// Mitsubishi GX Works2 project: PLC_Group5   PLC: FX3G

// global labels: Global1
VAR_GLOBAL
  Start_DAY AT X007 : BOOL;
  Lamp_Start_Internal AT M7 : BOOL;
END_VAR
VAR_GLOBAL CONSTANT
  Min_Protein : REAL := 320.0;
  Min_Oat : REAL := 400;
  Min_honey : REAL := 160.0;
END_VAR
VAR_GLOBAL
  End_Triger AT X005 : BOOL;
  End_Day AT M3 : BOOL;
  START_Day_Lamp AT X007 : BOOL;
  End_Day_Lamp AT X007 : BOOL;
  Lamp_Start_initaal AT M1 : BOOL;
  Day_Work_Lamp AT Y000 : BOOL;
  Mix_Products AT X003 : BOOL;
  Anlog_Inpute AT D8280 : INT;
END_VAR
VAR_GLOBAL CONSTANT
  Min_Analog : REAL := 5.0;
END_VAR
VAR_GLOBAL
  Save AT X007 : BOOL;
END_VAR
VAR_GLOBAL CONSTANT
  Max_Analog : REAL := 5;
END_VAR
VAR_GLOBAL
  Save_Anlog_Classic AT D8282 : INT;
  Save_Anlog_Protein AT D8282 : INT;
  Save_Lamp_Input AT M1 : BOOL;
END_VAR
VAR_GLOBAL CONSTANT
  Constant_400 : REAL := 400;
END_VAR
VAR_GLOBAL
  Normalized_Inpute AT M20 : BOOL;
  Input_Hone AT D1150 : REAL;
  M_hone AT D1152 : REAL;
  Input_Oat AT D1154 : REAL;
  M_Oat AT D1156 : REAL;
  Input_Protein AT D1158 : REAL;
  M_Protein AT D1160 : REAL;
  M_PM_Proteinrotein AT D1160 : REAL;
  Input_Ans AT D1302 : REAL;
  USER_PICK AT D1300 : REAL;
  Classic AT M22 : BOOL;
  Protein AT M23 : BOOL;
END_VAR
VAR_GLOBAL CONSTANT
  LessHone_120 : REAL := 120.0;
  LessOat_400 : REAL := 400.0;
  Less_Protien_160 : REAL := 160.0;
  LessOat_240 : REAL := 240.0;
  LessHone_160 : REAL := 160.0;
  LessProtien_320 : REAL := 320.0;
  LessHone_15 : REAL := 15.0;
  LessOat_50 : REAL := 50.0;
  Less_Protien_20 : REAL := 20.0;
  LessHone_20 : REAL := 20.0;
  LessOat_30 : REAL := 30.0;
  LessProtien_40 : REAL := 40.0;
END_VAR
VAR_GLOBAL
  Timer_MIX AT TC10 : BOOL;
END_VAR
VAR_GLOBAL CONSTANT
  Time_value : WORD := 50;
END_VAR
VAR_GLOBAL
  Lamp_MIX AT Y003 : BOOL;
  Start_baking AT X002 : BOOL;
  Blink_Lamp AT M30 : BOOL;
  Timer_Bake_Clasicc AT TC2 : BOOL;
END_VAR
VAR_GLOBAL CONSTANT
  Bakt_TimeClassic : WORD := 4;
END_VAR
VAR_GLOBAL
  Ts1 AT TC2 : BOOL;
  Baking_Lamp1 AT Y001 : BOOL;
  Timer_Bake_Protein AT TC3 : BOOL;
  Ts2 AT TC3 : BOOL;
  Baking_Lamp2 AT Y002 : BOOL;
  Start_packing AT X006 : BOOL;
  Add_Snack AT X000 : BOOL;
  Packing_Lamp AT Y004 : BOOL;
  Snack_Num AT CC1 : BOOL;
END_VAR
VAR_GLOBAL CONSTANT
  BOX : WORD := 1;
END_VAR
VAR_GLOBAL
  CS AT CS1 : BOOL;
  StoringSnacks AT X002 : BOOL;
END_VAR
VAR_GLOBAL CONSTANT
  Add_1 : REAL := 1.0;
  Div_analog2 : REAL := 40;
END_VAR
VAR_GLOBAL
  Num_of_Snacks_Packs AT D1202 : REAL;
  Analog_Output AT D8282 : INT;
  Protein_chose AT M23 : BOOL;
  Protein_chosen AT CC23 : BOOL;
  Classic_chosen AT CC22 : BOOL;
  Classic_1 AT M82 : BOOL;
  Protein_1 AT M89 : BOOL;
  Blinking_Lamp AT M33 : BOOL;
  Timer_Bake_One AT TC2 : BOOL;
  Timer_Bake_Two AT TC3 : BOOL;
END_VAR
VAR_GLOBAL CONSTANT
  TimeForCS : WORD := 30;
  TimeForPS : WORD := 60;
END_VAR
VAR_GLOBAL
  Flash_Count AT TC5 : BOOL;
  Bake_Time AT D5000 : WORD;
  CountFirst_Snack_Num AT CC1 : BOOL;
END_VAR
VAR_GLOBAL CONSTANT
  FirstBar : WORD := 1;
END_VAR
VAR_GLOBAL
  One_Bar_Count AT CS1 : BOOL;
  Seven_Bar_Count AT CS2 : BOOL;
  Count_7_bars AT CC2 : BOOL;
END_VAR
VAR_GLOBAL CONSTANT
  SevenBar : WORD := 8;
END_VAR
VAR_GLOBAL
  Snack_Storage AT D1202 : REAL;
  Stock_Check AT M50 : BOOL;
  StockStock_Check_Check AT M50 : BOOL;
END_VAR
VAR_GLOBAL CONSTANT
  ResAnalogOutput : INT;
  ZeroHone : REAL;
  ZeroOat : REAL;
  ZeroProtein : REAL;
END_VAR

// task Task_01 (event TRUE, interval 0, priority 31): POU_01

PROGRAM POU_01
(* structured ladder/FBD written out as ST: instructions are called as NAME(EN, inputs, outputs); _pN, _eN, _tN stand for wires *)
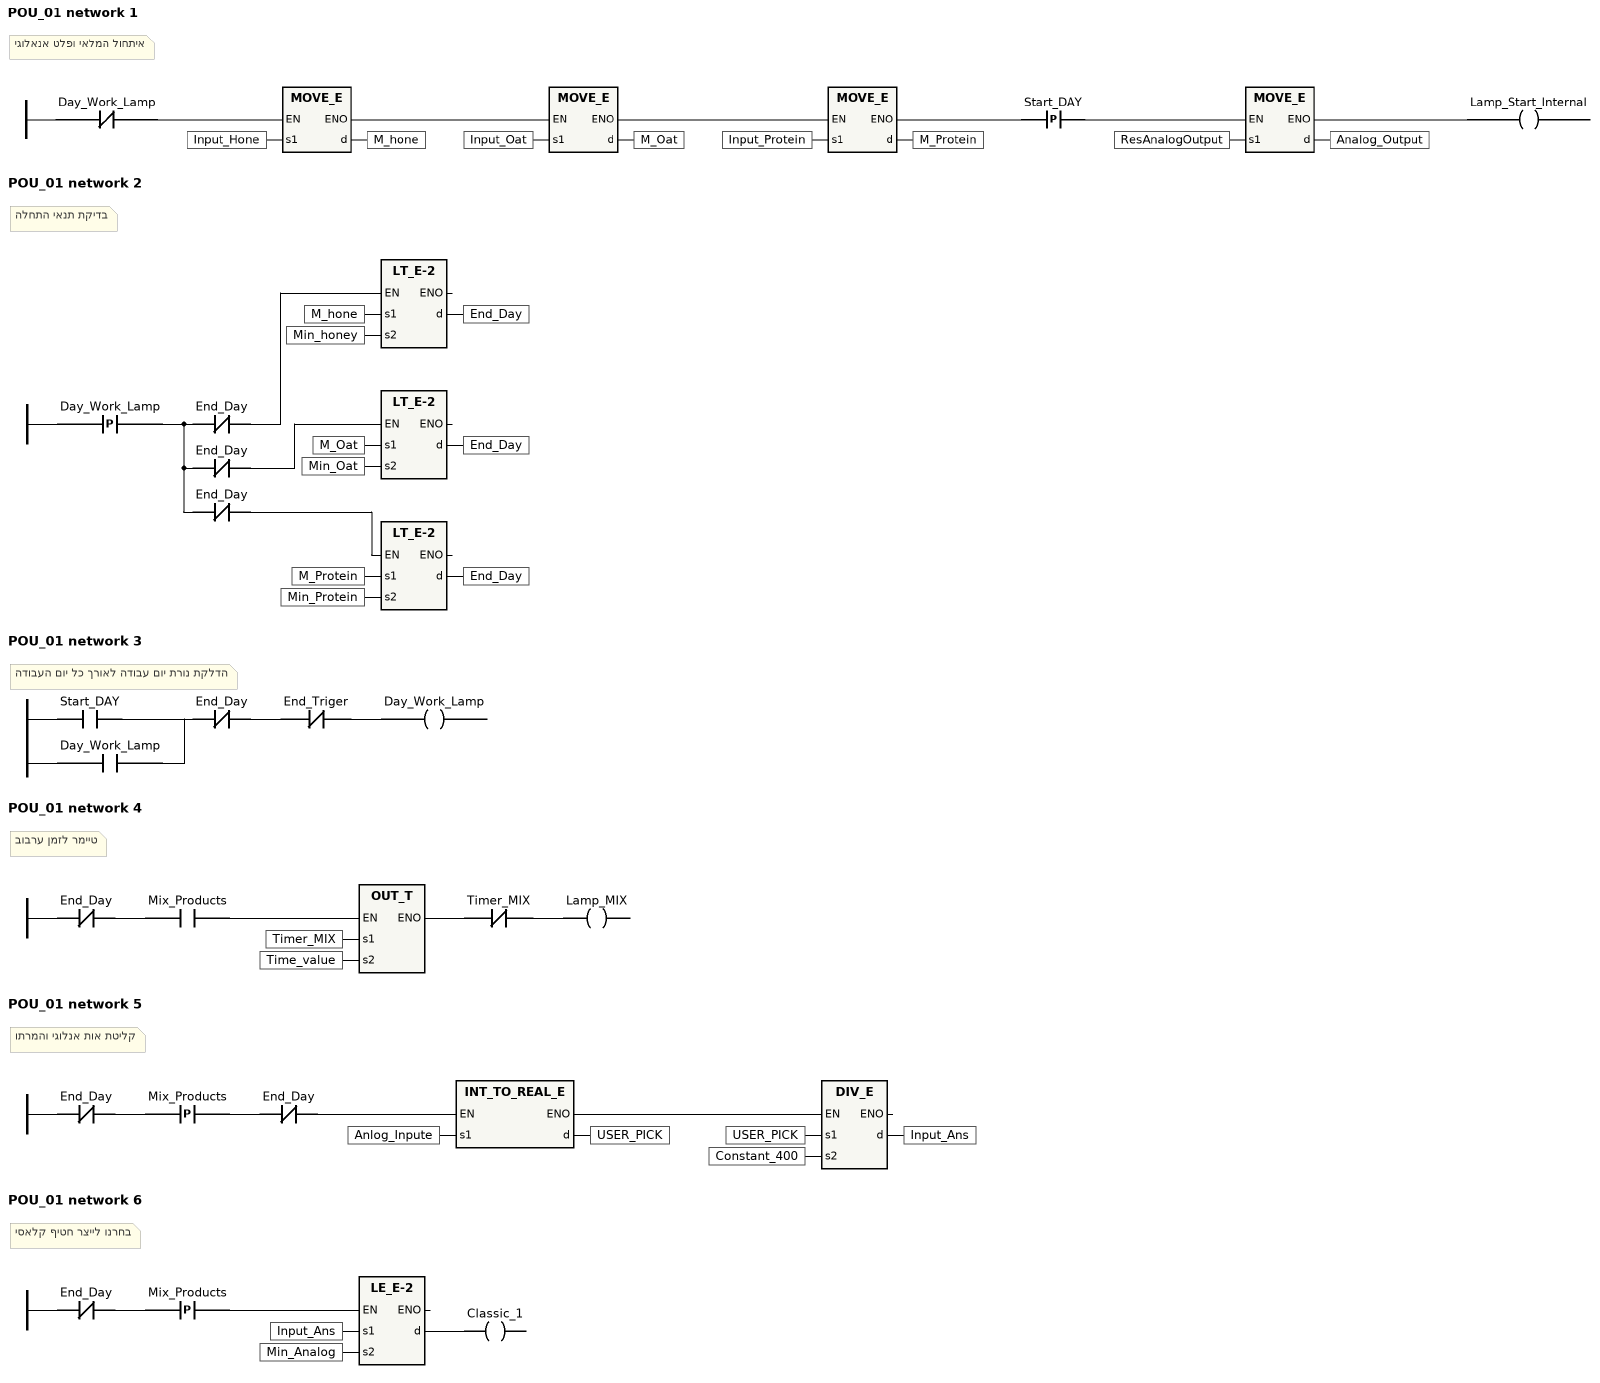
(* network 1 *)
(* איתחול המלאי ופלט אנאלוגי *)
_e1 := MOVE_E(NOT Day_Work_Lamp, Input_Hone, M_hone);
_e2 := MOVE_E(_e1, Input_Oat, M_Oat);
_e3 := MOVE_E(_e2, Input_Protein, M_Protein);
_e4 := MOVE_E(_e3 AND LDP(TRUE, Start_DAY), ResAnalogOutput, Analog_Output);
Lamp_Start_Internal := _e4;
(* network 2 *)
(* בדיקת תנאי התחלה *)
_p1 := LDP(TRUE, Day_Work_Lamp);
LT_E(_p1 AND NOT End_Day, M_hone, Min_honey, End_Day);
LT_E(_p1 AND NOT End_Day, M_Oat, Min_Oat, End_Day);
LT_E(_p1 AND NOT End_Day, M_Protein, Min_Protein, End_Day);
(* network 3 *)
(* הדלקת נורת יום עבודה לאורך כל יום העבודה *)
Day_Work_Lamp := ((Start_DAY OR Day_Work_Lamp) AND NOT End_Day) AND NOT End_Triger;
(* network 4 *)
(* טיימר לזמן ערבוב *)
_e1 := OUT_T(NOT End_Day AND Mix_Products, Timer_MIX, Time_value);
Lamp_MIX := _e1 AND NOT Timer_MIX;
(* network 5 *)
(* קליטת אות אנלוגי והמרתו *)
_e1 := INT_TO_REAL_E(NOT End_Day AND LDP(TRUE, Mix_Products) AND NOT End_Day, Anlog_Inpute, USER_PICK);
DIV_E(_e1, USER_PICK, Constant_400, Input_Ans);
(* network 6 *)
(* בחרנו לייצר חטיף קלאסי *)
LE_E(NOT End_Day AND LDP(TRUE, Mix_Products), Input_Ans, Min_Analog, _t1);
Classic_1 := _t1;
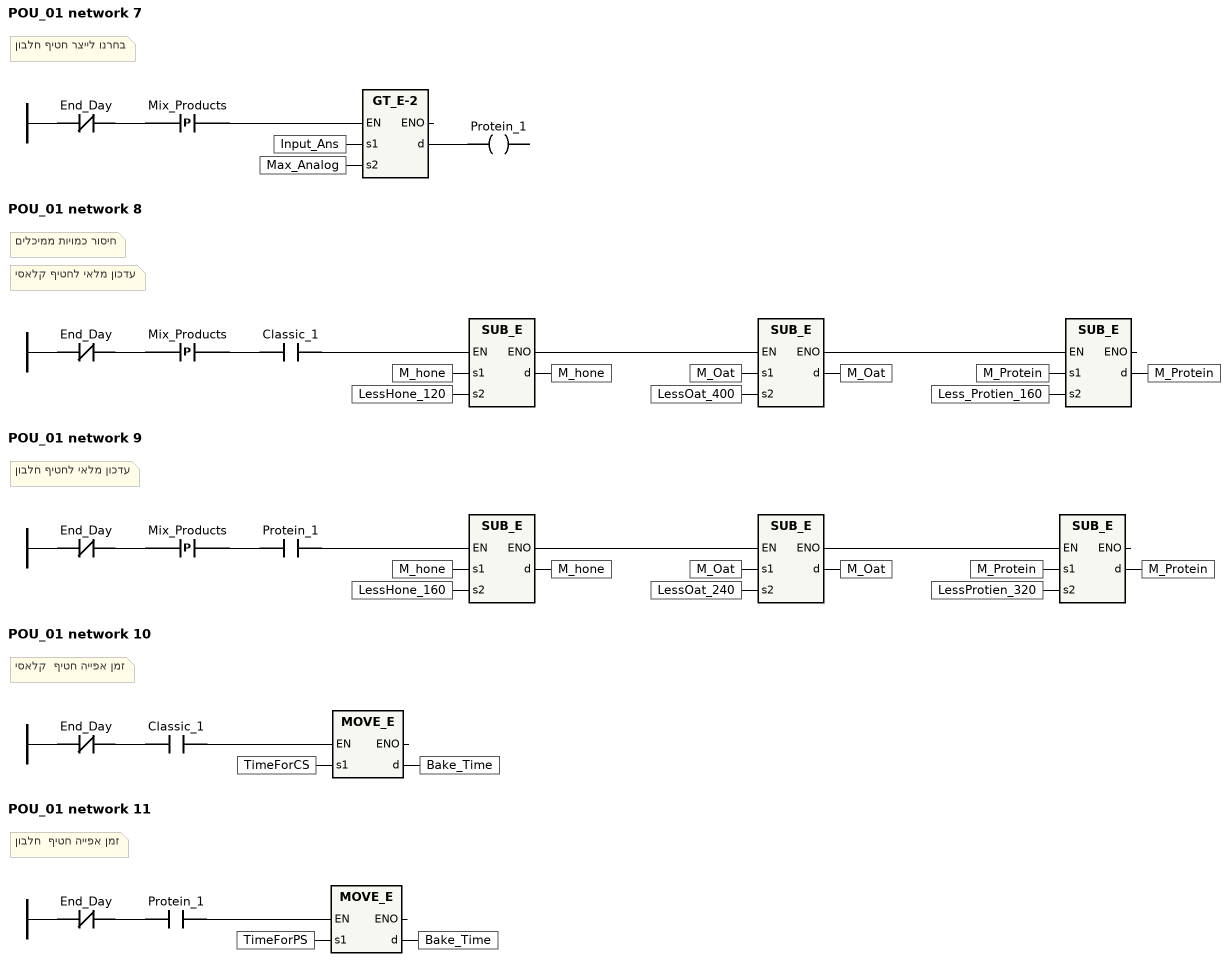
(* network 7 *)
(* בחרנו לייצר חטיף חלבון *)
GT_E(NOT End_Day AND LDP(TRUE, Mix_Products), Input_Ans, Max_Analog, _t1);
Protein_1 := _t1;
(* network 8 *)
(* חיסור כמויות ממיכלים *)
(* עדכון מלאי לחטיף קלאסי *)
_e1 := SUB_E(NOT End_Day AND LDP(TRUE, Mix_Products) AND Classic_1, M_hone, LessHone_120, M_hone);
_e2 := SUB_E(_e1, M_Oat, LessOat_400, M_Oat);
SUB_E(_e2, M_Protein, Less_Protien_160, M_Protein);
(* network 9 *)
(* עדכון מלאי לחטיף חלבון *)
_e1 := SUB_E(NOT End_Day AND LDP(TRUE, Mix_Products) AND Protein_1, M_hone, LessHone_160, M_hone);
_e2 := SUB_E(_e1, M_Oat, LessOat_240, M_Oat);
SUB_E(_e2, M_Protein, LessProtien_320, M_Protein);
(* network 10 *)
(* זמן אפייה חטיף  קלאסי *)
MOVE_E(NOT End_Day AND Classic_1, TimeForCS, Bake_Time);
(* network 11 *)
(* זמן אפייה חטיף  חלבון *)
MOVE_E(NOT End_Day AND Protein_1, TimeForPS, Bake_Time);
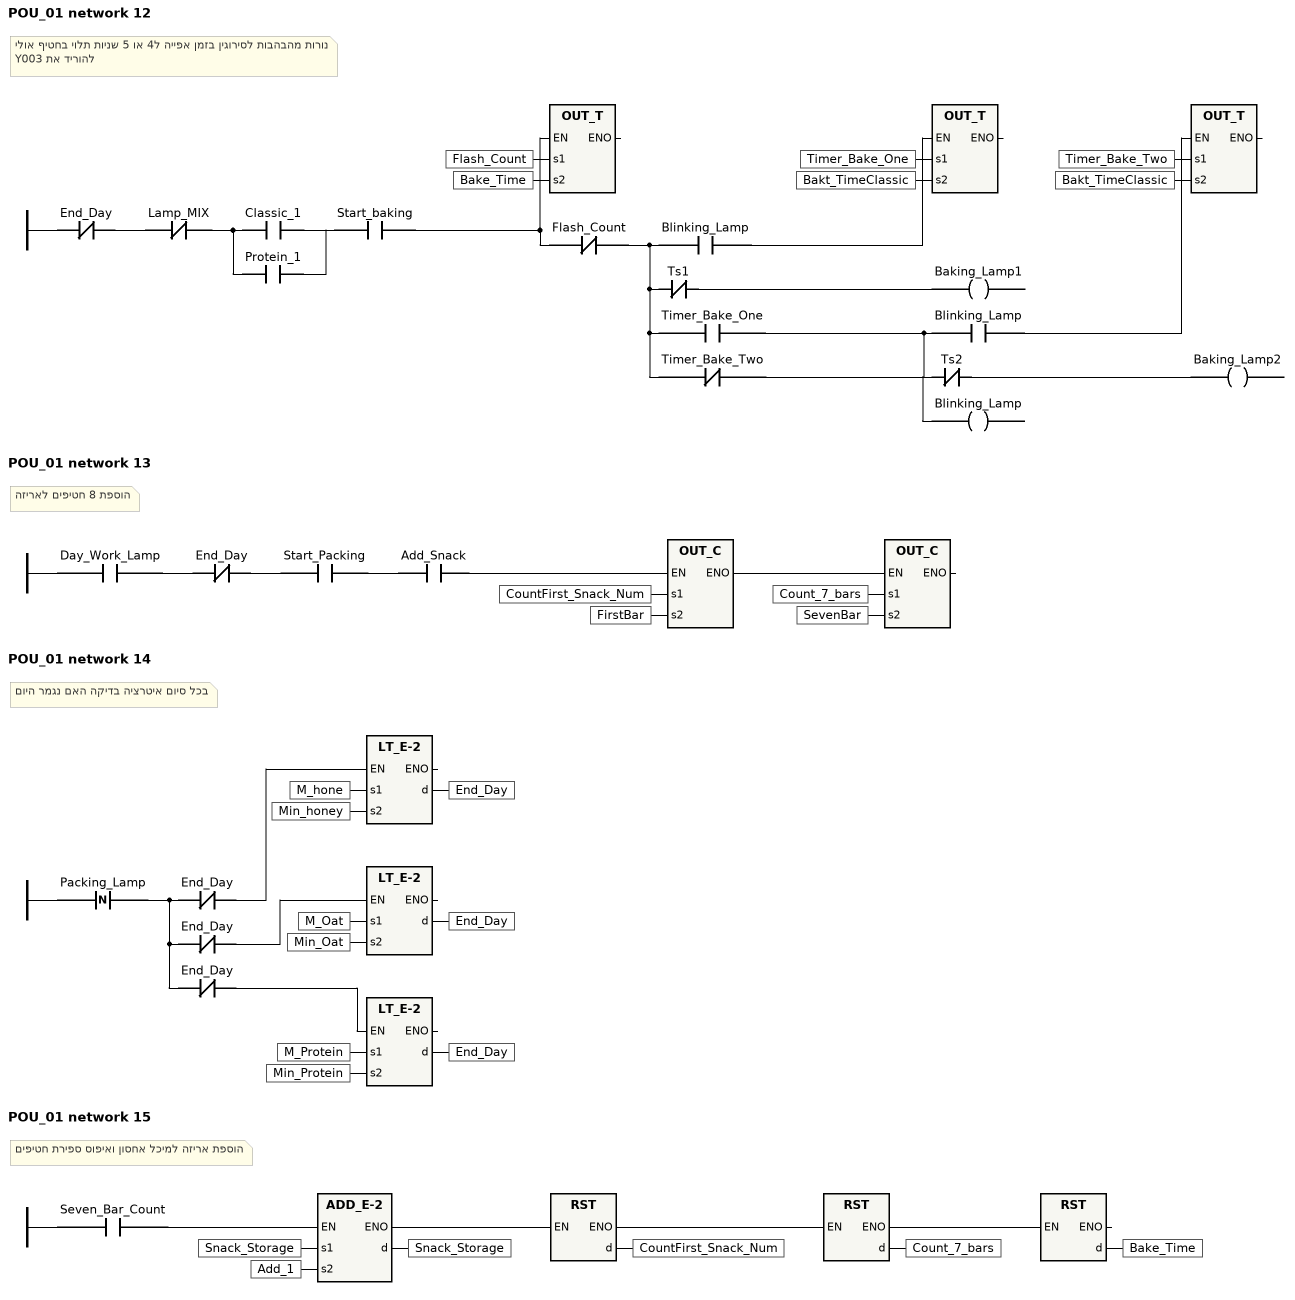
(* network 12 *)
(* נורות מהבהבות לסירוגין בזמן אפייה ל4 או 5 שניות תלוי בחטיף אולי להוריד את Y003 *)
_p1 := NOT End_Day AND NOT Lamp_MIX;
_p2 := ((_p1 AND Classic_1) OR (_p1 AND Protein_1)) AND Start_baking;
OUT_T(_p2, Flash_Count, Bake_Time);
_p3 := _p2 AND NOT Flash_Count;
OUT_T(_p3 AND Blinking_Lamp, Timer_Bake_One, Bakt_TimeClassic);
Baking_Lamp1 := _p3 AND NOT Ts1;
_p4 := _p3 AND Timer_Bake_One;
OUT_T(_p4 AND Blinking_Lamp, Timer_Bake_Two, Bakt_TimeClassic);
Baking_Lamp2 := _p4 AND NOT Ts2;
Blinking_Lamp := _p3 AND NOT Timer_Bake_Two;
(* network 13 *)
(* הוספת 8 חטיפים לאריזה *)
_e1 := OUT_C(Day_Work_Lamp AND NOT End_Day AND Start_Packing AND Add_Snack, CountFirst_Snack_Num, FirstBar);
OUT_C(_e1, Count_7_bars, SevenBar);
(* network 14 *)
(* בכל סיום איטרציה בדיקה האם נגמר היום *)
_p1 := LDF(TRUE, Packing_Lamp);
LT_E(_p1 AND NOT End_Day, M_hone, Min_honey, End_Day);
LT_E(_p1 AND NOT End_Day, M_Oat, Min_Oat, End_Day);
LT_E(_p1 AND NOT End_Day, M_Protein, Min_Protein, End_Day);
(* network 15 *)
(* הוספת אריזה למיכל אחסון ואיפוס ספירת חטיפים *)
_e1 := ADD_E(Seven_Bar_Count, Snack_Storage, Add_1, Snack_Storage);
_e2 := RST(_e1, CountFirst_Snack_Num);
_e3 := RST(_e2, Count_7_bars);
RST(_e3, Bake_Time);
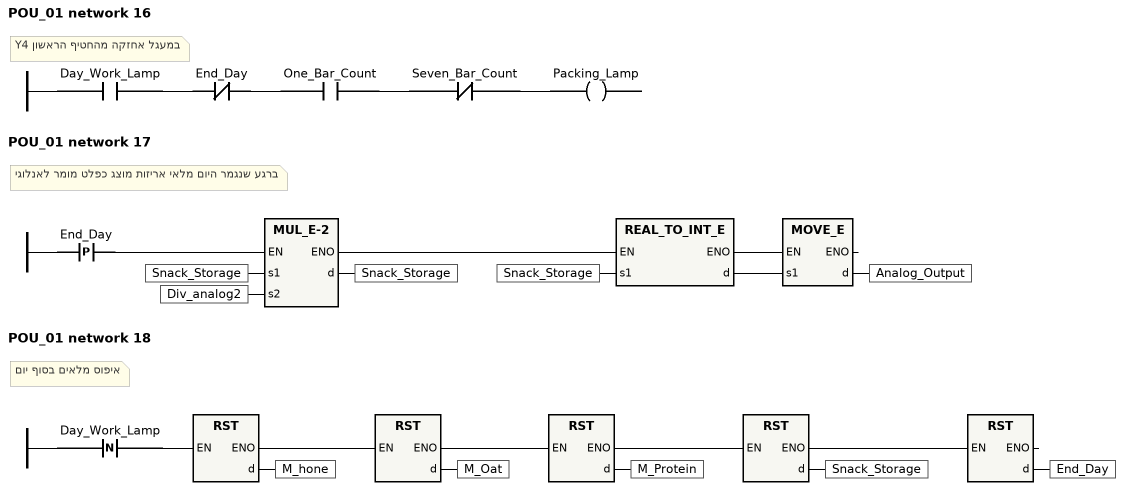
(* network 16 *)
(* Y4 במעגל אחזקה מהחטיף הראשון *)
Packing_Lamp := Day_Work_Lamp AND NOT End_Day AND One_Bar_Count AND NOT Seven_Bar_Count;
(* network 17 *)
(* ברגע שנגמר היום מלאי אריזות מוצג כפלט מומר לאנלוגי *)
_e1 := MUL_E(LDP(TRUE, End_Day), Snack_Storage, Div_analog2, Snack_Storage);
_e3 := REAL_TO_INT_E(_e1, Snack_Storage, _t2);
MOVE_E(_e3, _t2, Analog_Output);
(* network 18 *)
(* איפוס מלאים בסוף יום *)
_e1 := RST(LDF(TRUE, Day_Work_Lamp), M_hone);
_e2 := RST(_e1, M_Oat);
_e3 := RST(_e2, M_Protein);
_e4 := RST(_e3, Snack_Storage);
RST(_e4, End_Day);
END_PROGRAM
